// TIA Portal V18 export
DATA_BLOCK "PilzData"   // DB2702
{ S7_Optimized_Access := 'FALSE' }
VERSION : 0.1
// stored: AutoNumber false, DBAccessibleFromOPCUA true, DBAccessibleFromWebserver true, IsOnlyStoredInLoadMemory false, IsWriteProtectedInAS false
   VAR RETAIN
      "85A1" : Struct
         I8 : Bool;   // Light Current 1.1
         I9 : Bool;   // Light Current 1.2
         I10 : Bool;   // Light Current 2.1
         I11 : Bool;   // Light Current 2.2
         I12 : Bool;   // Stove E Stop_2.1
         I13 : Bool;   // Stove E Stop_2.2
         I14 : Bool;   // E Stop Feedback
         I15 : Bool;   // Safety Gate Feedback
         I0 : Bool;   // Control On
         I1 : Bool;   // Control Off
         I2 : Bool;   // Spare
         I3 : Bool;   // Spare
         I4 : Bool;   // E Stop_1.1
         I5 : Bool;   // E Stop_1.2
         I6 : Bool;   // Safety Gate 1.1
         I7 : Bool;   // Safety Gate 1.2
         I24 : Bool;
         I25 : Bool;
         I26 : Bool;
         I27 : Bool;
         I28 : Bool;
         I29 : Bool;
         I30 : Bool;
         I31 : Bool;
         I16 : Bool;   // Light Current 1 feedback
         I17 : Bool;   // Light Current 2 feedback
         I18 : Bool;   // Stove E Stop feedback
         I19 : Bool;   // Spare
         I20 : Bool;   // I20
         I21 : Bool;   // I21
         I22 : Bool;   // I22
         I23 : Bool;   // I23
         O0 : Bool;
         O1 : Bool;
         O2 : Bool;
         O3 : Bool;
         Spare_1 : Bool;
         Spare_2 : Bool;
         Spare_3 : Bool;
         Spare_4 : Bool;
         Spare_5 : Bool;
         Spare_6 : Bool;
         Spare_7 : Bool;
         Spare_8 : Bool;
         Spare_9 : Bool;
         Spare_10 : Bool;
         Spare_11 : Bool;
         Spare_12 : Bool;
      END_STRUCT;
      "85A2" : Struct
         I0 : Bool;   // UnLoadingMaterialDoor 1.1
         I1 : Bool;   // UnLoadingMaterialDoor 1.2
         I2 : Bool;   // UnLoadingMaterialDoor 2.1
         I3 : Bool;   // UnLoadingMaterialDoor 2.2
         I4 : Bool;   // UnLoadingMaterialDoor 3.1
         I5 : Bool;   // UnLoadingMaterialDoor 3.2
         I6 : Bool;   // LoadingMaterialDoor 4.1
         I7 : Bool;   // LoadingMaterialDoor 4.2
         O0 : Bool;
         O1 : Bool;
         O2 : Bool;
         O3 : Bool;
         Spare_1 : Bool;
         Spare_2 : Bool;
         Spare_3 : Bool;
         Spare_4 : Bool;
      END_STRUCT;
      "85A3" : Struct
         I0 : Bool;   // MaterialDoor 1 feedback
         I1 : Bool;   // MaterialDoor 2 feedback
         I2 : Bool;   // MaterialDoor 3 feedback
         I3 : Bool;   // MaterialDoor 4 feedback
         I4 : Bool;   // Stove Door feedback 1.1
         I5 : Bool;   // Stove Door feedback 1.2
         I6 : Bool;   // Robot feedback
         I7 : Bool;   // Robot Door feedback
         O0 : Bool;
         O1 : Bool;
         O2 : Bool;
         O3 : Bool;
         Spare_1 : Bool;
         Spare_2 : Bool;
         Spare_3 : Bool;
         Spare_4 : Bool;
      END_STRUCT;
      "85A4" : Struct
         I0 : Bool;   // LoadingMaterialDoor 1.1
         I1 : Bool;   // LoadingMaterialDoor 1.2
         I2 : Bool;   // LoadingMaterialDoor 2.1
         I3 : Bool;   // LoadingMaterialDoor 2.2
         I4 : Bool;   // LoadingMaterialDoor 3.1
         I5 : Bool;   // LoadingMaterialDoor 3.2
         I6 : Bool;   // NG 2 Door 1.1
         I7 : Bool;   // NG 2 Door 1.2
         O0 : Bool;
         O1 : Bool;
         O2 : Bool;
         O3 : Bool;
         Spare_1 : Bool;
         Spare_2 : Bool;
         Spare_3 : Bool;
         Spare_4 : Bool;
      END_STRUCT;
      "85A5" : Struct
         I0 : Bool;   // Robot 1 E Stop1.1
         I1 : Bool;   // Robot 1 E Stop1.2
         I2 : Bool;   // Robot 2 E Stop1.1
         I3 : Bool;   // Robot 2 E Stop1.2
         I4 : Bool;   // Robot 3 E Stop1.1
         I5 : Bool;   // Robot 3 E Stop1.2
         I6 : Bool;   // NG 1 Door 1.1
         I7 : Bool;   // NG 1 Door 1.2
         O0 : Bool;
         O1 : Bool;
         O2 : Bool;
         O3 : Bool;
         Spare_1 : Bool;
         Spare_2 : Bool;
         Spare_3 : Bool;
         Spare_4 : Bool;
      END_STRUCT;
      TON { S7_SetPoint := 'True'} : Array[0..50] of TON_TIME;
      OK_BoxFlag : Struct
         X_Moving : Bool;
         Y_Pulling : Bool;
         X_Need_MoveBox : Bool;
         Y_Need_PullBox : Bool;
         Pushing : Bool;
         ChangeUnloadingBox : Bool;
         HMIChangeUnloadingBox : Bool;
         ManualOKBox : Bool;
         HMIManualOKBox : Int;
      END_STRUCT;
      Status : Int;
   END_VAR
BEGIN
END_DATA_BLOCK
